SUBAPPLICATION Uebung_010c2 (* SoftKey_F1 auf DigitalOutput_Q1 mit GreenWhiteBackground mit Subapp *)
  (* Standard: 61499-2; Description: Copyright (c) 2023 Meisterschulen am Ostbahnhof This program and the accompanying materials are made available under the terms of the Eclipse Public License 2.0 which is available at https://www.eclipse.org/legal/epl-2.0/ SPDX-License-Identifier: EPL-2.0 *)
  (* Version 1.0, 2023-10-23, Franz Höpfinger, Meisterschulen am Ostbahnhof *)
  PACKAGE Uebungen;
  IMPORT Uebungen::const::UT::DefaultPool::SoftKey_F1;
  IMPORT logiBUS::io::DQ::logiBUS_DO;
  IMPORT logiBUS::io::DQ::logiBUS_DO_S;
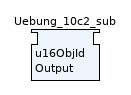
  SUBAPPLICATION Uebung_10c2_sub
    VAR_INPUT
      u16ObjId : UINT := SoftKey_F1; (* Object ID *)
      Output : logiBUS::io::DQ::logiBUS_DO_S := logiBUS_DO::Output_Q1; (* Identify the Output Output_Q1..Q8 *)
    END_VAR
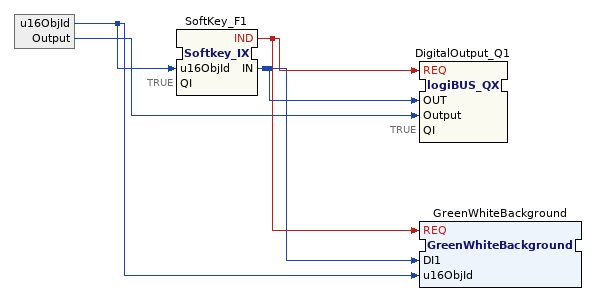
    FBS
      DigitalOutput_Q1 : logiBUS::io::DQ::logiBUS_QX(QI := TRUE);
      SoftKey_F1 : isobus::UT::io::Softkey::Softkey_IX(QI := TRUE);
    END_FBS
    SUBAPPS
      GreenWhiteBackground : Uebungen::sys::GreenWhiteBackground;
    END_SUBAPPS
    EVENT_CONNECTIONS
      SoftKey_F1.IND TO GreenWhiteBackground.REQ;
      SoftKey_F1.IND TO DigitalOutput_Q1.REQ;
    END_CONNECTIONS
    DATA_CONNECTIONS
      SoftKey_F1.IN TO GreenWhiteBackground.DI1;
      SoftKey_F1.IN TO DigitalOutput_Q1.OUT;
      u16ObjId TO SoftKey_F1.u16ObjId;
      u16ObjId TO GreenWhiteBackground.u16ObjId;
      Output TO DigitalOutput_Q1.Output;
    END_CONNECTIONS
  END_SUBAPPLICATION
END_SUBAPPLICATION
